# EPICS autosave request: iocBoot/iocNoiseSrc/auto_settings_noiseSrc.req
file "noiseSrc_settings.req",                P=$(P),  R=$(R)
